// TIA Portal V20 export
DATA_BLOCK "Q_DAS_DB"   // DB102
// stored: InstanceOfName Unit1.Q_DAS, InstanceOfType FB, Namespace Unit1
"Unit1.Q_DAS"
   // VAR
   //    m1 : Bool;
   // END_VAR
BEGIN
END_DATA_BLOCK
